(*********************************** G.D S.p.A. - Technical Department ***********************************
============= PROGRAM INFO ============
FOLDER:             TBD
MACHINES INVOLVED:  TBD 

============= DESCRIPTION =============

============= REVISIONS ===============
Date		Version	 	Author      	Description             
----------	-------		------------  	--------------------------------------------
2019/04/24 	0000.00	 	M.Grasso		Creation of the PRG

**********************************************************************************************************)
(*$R 
	process_ref:= prc; 
$*)
PROGRAM csp_case_main_safety_drives
VAR
	prc:					process;
	prc_path:				STRING;	
END_VAR

_read_var_input();

_objects_manager();

IF NOT objects_running()
THEN
	RETURN;	
END_IF

_read_process_image();

_mode_manager();

CASE process_get_mode(prc) OF
	MODE_ABSENT,
	MODE_INACTIVE:
		RETURN;
	MODE_TEST:
		;
END_CASE

_set_runtime_properties();

(********************************* BODY *********************************)

(************************************************************************)

_handle_messages();

_write_output();

ACTION _handle_messages:
;
END_ACTION

ACTION _handle_process_test:
;
END_ACTION

ACTION _mode_manager:
IF process_mode_req_is_pending(prc)
THEN
    process_apply_mode_req_first_step(prc);
    CASE process_get_mode(prc) OF
        MODE_TO_ABSENT:
			;
        MODE_TO_INACTIVE:
			;
        MODE_TO_TEST:
			;
        MODE_TO_OPERATIONAL:
			;
    END_CASE
    process_apply_mode_req_second_step(prc);
END_IF
END_ACTION

ACTION _objects_manager:
IF objects_initialization()
THEN
	sub_process_init(
		object_name					:= 'csp_case_main_safety_drives.prc', 
		process						:= csp_case_main_safety.prc, 
		CONVERSION_this				:= prc);
		
	prc_path 						:= process_get_path(prc);		
END_IF

IF objects_running()
THEN
	process_cycle(prc);
END_IF
END_ACTION

ACTION _read_process_image:
;
END_ACTION

ACTION _read_var_input:
;
END_ACTION

ACTION _set_runtime_properties:
;
END_ACTION

ACTION _write_output:
;
END_ACTION

END_PROGRAM

(* stored: Version 1.1.0.1, ProductVersion 3.1.4022.12
   POU csp_case_main_safety_drives: Id {d5ba84e7-2d4e-4dad-bec6-7108bba56e37}, SpecialFunc None
   Action _handle_messages: Id {d08a2bf0-179c-4816-a708-05be8e5791ea}
   Action _handle_process_test: Id {bb766444-6c9e-4704-96a4-6faecb5160f8}
   Action _mode_manager: Id {64409300-4b33-42ee-befd-8f6e8fecf583}
   Action _objects_manager: Id {0ccf9d81-da90-42fd-9660-bc50f4d05381}
   Action _read_process_image: Id {6c59dda0-7547-4e5c-9726-38d20bc5e3a5}
   Action _read_var_input: Id {0b46747d-dff5-4aa6-9869-f16de8310c2a}
   Action _set_runtime_properties: Id {652c59a8-e1ad-4536-ae31-d9b6eb7d1151}
   Action _write_output: Id {097ded47-fe49-46c5-9e62-5e9f74704e99} *)
